// TIA Portal V16 export
// export: Created 2021-04-11T09:51:21.442573Z, ExportSetting WithDefaults, DisplayName Totally Integrated Automation Portal, DisplayVersion V16, DisplayName TIA Portal Version Control Interface, DisplayVersion V16, DisplayName TIA Portal Openness, DisplayVersion V16, DisplayName STEP 7 Professional, DisplayVersion V16, DisplayName STEP 7 Safety, DisplayVersion V16, DisplayName WinCC Unified SCADA Engineering System, DisplayVersion V16
FUNCTION_BLOCK "controlValve"   // FB2, LAD
{ S7_Optimized_Access := 'TRUE' }
VERSION : 0.1
// stored: AutoNumber true, IsIECCheckEnabled false, IsRetainMemResEnabled false, MemoryReserve 100, SetENOAutomatically false, UDAEnableTagReadback false
   VAR_INPUT
      autoclose_M : Bool;   // режим автозакрытия
      time_autoclose : Time := T#2000ms;
      "time_open/close" : Time := T#2000ms;
   END_VAR
   VAR_OUTPUT
      openQ : Bool;   // катушка на открытие
      closeQ : Bool;   // катушка на закрытие
   END_VAR
   VAR_IN_OUT
      open : Bool;   // сигнал на открытие
      close : Bool;   // сигнал на закрытие
      stopAlarm : Bool;   // сигнал резкого выключения
   END_VAR
   VAR
      tofOpen : TOF_TIME;   // время в течении которого катушка на открытие включена
      tofClose : TOF_TIME;   // время в течении которого катушка на закрытие включена
      Ptrig : Array[0..1] of Bool;   // триггеры ловят импульсный сигнал о включении и выключении
      Ntrig : Array[0..1] of Bool;
      tonAutoclose_M : TON_TIME;   // время через которое сработает автозакрытие
   END_VAR
   VAR_TEMP   // added for the SCL form of the ladder/FBD networks
      _w1 : Bool;
      _w2 : Bool;
      _w3 : Bool;
      _w4 : Bool;
      _w5 : Bool;
      _w6 : Bool;
   END_VAR
BEGIN

REGION Network 1: сигнал на открытие
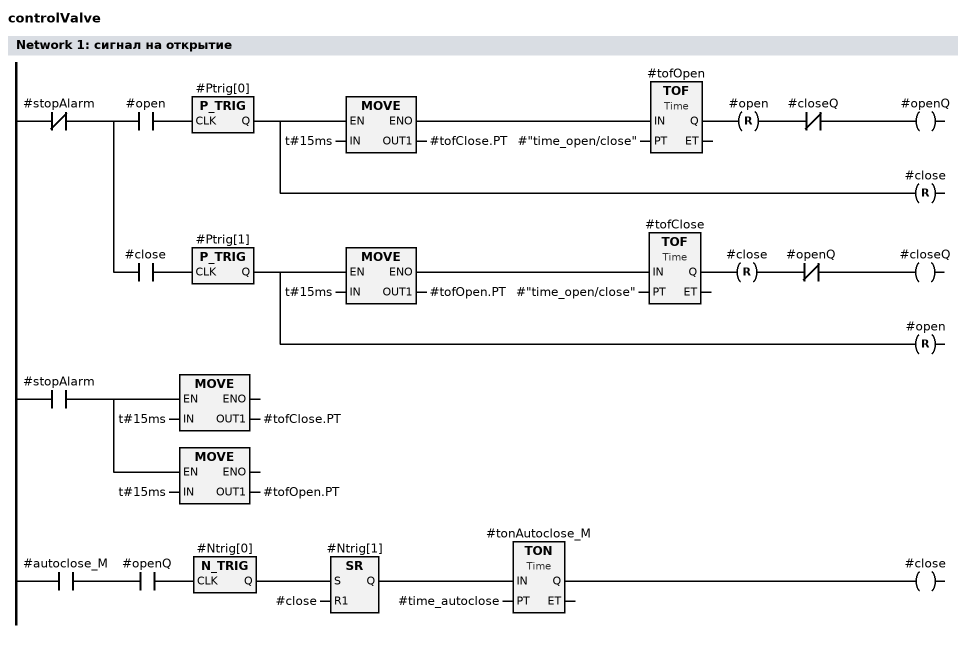
   RUNG wire#powerrail
      I_Contact( #stopAlarm )
      wire#w1
      Contact( #open )
      P_Trig( #Ptrig[0] )
      wire#w2
      Move(in := t#15ms, out1 => #tofClose.PT)
      { S7_Templates := "time_type := Time" } #tofOpen.TOF(pt := #"time_open/close", et =>)
      R_Coil( #open )
      I_Contact( #closeQ )
      Coil( #openQ )
   END_RUNG
   RUNG wire#w2
      R_Coil( #close )
   END_RUNG
   RUNG wire#w1
      Contact( #close )
      P_Trig( #Ptrig[1] )
      wire#w3
      Move(in := t#15ms, out1 => #tofOpen.PT)
      { S7_Templates := "time_type := Time" } #tofClose.TOF(pt := #"time_open/close", et =>)
      R_Coil( #close )
      I_Contact( #openQ )
      Coil( #closeQ )
   END_RUNG
   RUNG wire#w3
      R_Coil( #open )
   END_RUNG
   RUNG wire#powerrail
      Contact( #stopAlarm )
      wire#w4
      Move(in := t#15ms, out1 => #tofClose.PT)
   END_RUNG
   RUNG wire#w4
      Move(in := t#15ms, out1 => #tofOpen.PT)
   END_RUNG
   RUNG wire#powerrail
      Contact( #autoclose_M )
      Contact( #openQ )
      N_Trig( #Ntrig[0] )
      S_SR(operand := #Ntrig[1], r1 := #close)
      { S7_Templates := "time_type := Time" } #tonAutoclose_M.TON(pt := #time_autoclose, et =>)
      Coil( #close )
   END_RUNG
   // the same network as SCL:
   #_w1 := NOT #stopAlarm AND #open;
   #_w2 := #_w1 AND NOT #Ptrig[0];   // rising edge
   #Ptrig[0] := #_w1;
   IF #_w2 THEN #tofClose.PT := t#15ms; END_IF;
   #tofOpen(IN := #_w2, PT := #"time_open/close");   // TOF
   IF #tofOpen.Q THEN #open := FALSE; END_IF;
   #openQ := #tofOpen.Q AND NOT #closeQ;
   IF #_w2 THEN #close := FALSE; END_IF;
   #_w3 := NOT #stopAlarm AND #close;
   #_w4 := #_w3 AND NOT #Ptrig[1];   // rising edge
   #Ptrig[1] := #_w3;
   IF #_w4 THEN #tofOpen.PT := t#15ms; END_IF;
   #tofClose(IN := #_w4, PT := #"time_open/close");   // TOF
   IF #tofClose.Q THEN #close := FALSE; END_IF;
   #closeQ := #tofClose.Q AND NOT #openQ;
   IF #_w4 THEN #open := FALSE; END_IF;
   IF #stopAlarm THEN
       #tofClose.PT := t#15ms;
       #tofOpen.PT := t#15ms;
   END_IF;
   #_w5 := #autoclose_M AND #openQ;
   #_w6 := NOT #_w5 AND #Ntrig[0];   // falling edge
   #Ntrig[0] := #_w5;
   IF #_w6 THEN
       #Ntrig[1] := TRUE;   // SR flip-flop
   END_IF;
   IF #close THEN #Ntrig[1] := FALSE; END_IF;
   #tonAutoclose_M(IN := #Ntrig[1], PT := #time_autoclose);   // TON
   #close := #tonAutoclose_M.Q;
END_REGION
END_FUNCTION_BLOCK
